Staubli VAL3: Transmission.pgx

program Transmission()
  local num nByteOut[48]
  local num nTranC[6]
begin
  nTranC[0]=shere[0].trsf.x
  nTranC[1]=shere[0].trsf.y
  nTranC[2]=shere[0].trsf.z
  nTranC[3]=shere[0].trsf.rx
  nTranC[4]=shere[0].trsf.ry
  nTranC[5]=shere[0].trsf.rz
  toBinary(nTranC,6,"8.0b",nByteOut)
  sioSet(sSocketout,nByteOut)
end
